INTERFACE ISumCollectorLINT EXTENDS CNM_AbstractObject.IObject

METHOD addValue
VAR_INPUT
	value :LINT;
END_VAR
END_METHOD

PROPERTY enabled : BOOL
GET
END_GET
SET
END_SET
END_PROPERTY

PROPERTY sum : LINT
GET
END_GET
SET
END_SET
END_PROPERTY

END_INTERFACE

(* stored: Version 1.1.0.1
   Itf ISumCollectorLINT: Id {63a5dcea-26bc-4d33-9956-e97b3e1c003c}
   Method addValue: Id {6ce63ed9-cec4-493f-9f2a-232d8d238cfe}
   Property enabled: Id {8af8e446-90cc-4712-8d12-640844d5690e}
   Get Get: Id {32225075-ece5-4e84-980a-93d7ab28fdcf}
   Set Set: Id {676a8b64-50bd-4e4e-9ee1-aab7253a5cb7}
   Property sum: Id {a64c9fc2-087c-4f1d-a724-1410d388d488}
   Get Get: Id {8e137847-8821-4b1c-a417-a01b27772185}
   Set Set: Id {53963f74-8a19-4975-8d36-27043b1553f2} *)
